TYPE ST_PhasingAbsParams :
STRUCT
	PhaseShift		: LREAL;
	Velocity		: LREAL;
	Acceleration	: LREAL;
	Deceleration	: LREAL;
	Jerk			: LREAL;
END_STRUCT
END_TYPE

(* stored: Version 1.1.0.1, ProductVersion 3.1.4023.8
   DUT ST_PhasingAbsParams: Id {1c284bfe-17e7-4573-badf-df834ecc27be} *)
